FUNCTION_BLOCK SensorFQM
VAR_INPUT
END_VAR
VAR_OUTPUT
END_VAR
VAR_IN_OUT
	
END_VAR
VAR
	State:VisionState:= 0;
	SensorToPlc AT %I*:SensorToPlc;
	PlcToSensor AT %Q*:PlcToSensor;
	KeepAliveTimer:TON;
	
	RExec:R_TRIG;
	NextCycleResetFlags:BOOL;
	Results: ARRAY [0..7] OF REAL;
	
	//Single measurement
	RequestSingle:BOOL;
	TakePhoto:BOOL;
	TakePhotoFlag:R_TRIG;
	MeasureTimer:TON;
	MeasureTime:TIME;
	
	//Continuous measurement
	RequestStartCont:BOOL;
	RequestStopCont:BOOL;
	StopFromError:BOOL;
	ResponseTimer:TON;
	ResponseTime:TIME;
	FEnable:F_TRIG;
	
	LastResult:INT:=0;//0-Null, 1-Ok, 2-NG
	
	//Error Management
	RequestErrorCode:BOOL;
	LastError:DWORD;
END_VAR
VAR CONSTANT
	KeepAliveBit:INT:=24;
END_VAR

// Preparing Inputs
SensorToPlc.FLG:= SensorToPlc.VisionStatusFlag.0;
SensorToPlc.BUSY:= SensorToPlc.VisionStatusFlag.1;
SensorToPlc.READY:= SensorToPlc.VisionStatusFlag.2;
SensorToPlc.OR_Jud:= SensorToPlc.VisionStatusFlag.3;
SensorToPlc.RUN:= SensorToPlc.VisionStatusFlag.4;
SensorToPlc.ERR:= SensorToPlc.VisionStatusFlag.15;
SensorToPlc.GATE:= SensorToPlc.VisionStatusFlag.16;
//Change a bit every 500ms as Keep Alive bit
(*KeepAliveTimer(in:=NOT KeepAliveTimer.Q, pt:=T#1S);
IF KeepAliveTimer.Q THEN
	PlcToSensor.VisionControlFlag.24:= NOT PlcToSensor.VisionControlFlag.24;
END_IF*)

//Delete variables. Estado distinto de 999 para permitir modificar a mano en ese estado especial
IF State <> 999 THEN
	PlcToSensor.EXE:=FALSE;
	PlcToSensor.ERCLR:=FALSE;
	PlcToSensor.DSA:=FALSE;
	PlcToSensor.TRIG:=FALSE;
END_IF

//State machine
CASE State OF
	000: //Error. Por ahora se salta parada cuando hay error
		IF NOT SensorToPlc.ERR THEN
			State := 010;
		ELSE
			State := 001;
		END_IF
			
	001: //Checking errors
		//TODO: Revisar
		_prepareCommand(Command:= VisionCmd.GetLatestError);
		PlcToSensor.EXE := TRUE;
		IF SensorToPlc.FLG THEN
			PlcToSensor.EXE := FALSE;
			LastError:= SensorToPlc.VisionResponseData;
			State := 002;
		END_IF
	002: //Clear data
		_prepareCommand(VisionCmd.ClearDataOutputBuffer);
		PlcToSensor.EXE := TRUE;
		IF SensorToPlc.FLG THEN
			PlcToSensor.EXE := FALSE;
			State := 003;
		END_IF
	003: //Clear Error
		PlcToSensor.ERCLR:=TRUE;
		IF NOT SensorToPlc.ERR THEN
			PlcToSensor.ERCLR := FALSE;
			State := 010;
		END_IF
	010: //StandStill
		IF RequestSingle THEN
			LastError := 0; //Elimina ultimo error cuando se pasa a este estado
			State := 011;
		END_IF
		IF RequestStartCont AND NOT RequestSingle THEN
			State := 012;
		END_IF
		IF SensorToPlc.ERR THEN
			State := 001;
			
		END_IF
	011: //Switching to Single
		_prepareCommand(VisionCmd.StartSingle);
		PlcToSensor.EXE:=TRUE;
		IF SensorToPlc.FLG THEN
			PlcToSensor.EXE := FALSE;
			State := 030;
			LastResult:=0;
		END_IF
	012: //Switching to continuous
		_prepareCommand(VisionCmd.StartContinuous);
		PlcToSensor.EXE:=TRUE;
		IF SensorToPlc.FLG THEN
			PlcToSensor.EXE := FALSE;
			State := 020;
		END_IF
	020: //Continuous Measurement
		//Loop to request measurement
		IF SensorToPlc.GATE THEN
			ResponseTime:=ResponseTimer.ET;
			PlcToSensor.DSA := FALSE;
			ResponseTimer(in:=FALSE, pt:=T#10S);
		ELSIF NOT SensorToPLC.gate THEN
			ResponseTimer(in:=TRUE, pt:=T#10S);
			PlcToSensor.DSA := TRUE;
		END_IF
		//transitions
		IF SensorToPLC.ERR THEN
			PlcToSensor.EXE := FALSE;
			StopFromError:=TRUE;
			State := 021;
		END_IF 
		IF RequestStopCont THEN
			PlcToSensor.EXE := FALSE;
			State := 021;
		END_IF
	021: //Stopping continuous
	    _prepareCommand(VisionCmd.StopContinuous);
		PlcToSensor.EXE := TRUE;
		IF SensorToPLC.FLG THEN
			IF StopFromError THEN
				PlcToSensor.EXE :=FALSE;
				StopFromError:=FALSE;
				State := 001;
			ELSE
				State := 010;
			END_IF
			RequestStopCont := FALSE;
		END_IF
	030: // Single Measurement Ready
		
		IF TakePhoto THEN
			//Take photo and request
			PlcToSensor.TRIG:=TRUE;
			PlcToSensor.DSA:=TRUE;
			MeasureTimer(in:=FALSE);
			MeasureTimer(in:=TRUE, pt:=T#60s);
			State := 31;
		END_IF
		IF NOT RequestSingle THEN
			State := 010;
		END_IF
		IF SensorToPlc.ERR THEN
			State := 001;
			_prepareCommand(Command:= VisionCmd.GetLatestError);
			PlcToSensor.EXE := TRUE;
		END_IF
	031: // Single Measurement Taking photo
		PlcToSensor.DSA := TRUE; // Ojo, ya se activo en el ciclo anterior. no hay retardo de un ciclo.
		PlcToSensor.TRIG := TRUE;
		MeasureTimer(in:=TRUE);
		IF SensorToPLC.GATE THEN
			//TODO: Esto llega mas tarde que el dato. Revisar.
			IF SensorToPlc.OR_Jud THEN
				LastResult:=2;
			ELSE
				LastResult:=1;
			END_IF
			MeasureTime:=MeasureTimer.ET;
			MeasureTimer(in:=FALSE);
			State := 030;
			PlcToSensor.TRIG:=FALSE;
			PlcToSensor.DSA:=FALSE;
		END_IF
		IF SensorToPLC.ERR THEN
			State := 001;
		END_IF
END_CASE

//Update Flag Bits into DWORD
PlcToSensor.VisionControlFlag.0:= PlcToSensor.EXE;
PlcToSensor.VisionControlFlag.1:= PlcToSensor.TRIG;
PlcToSensor.VisionControlFlag.15:= PlcToSensor.ERCLR;
PlcToSensor.VisionControlFlag.16:= PlcToSensor.DSA;

METHOD PRIVATE _prepareCommand
VAR_INPUT
	Command:VisionCmd;
END_VAR
VAR
	
END_VAR
(* 
Command orders deliverable to camera.
See OMRON FQ-M Series Vision Sensor docs for information
*)
CASE Command OF
	VisionCmd.StartSingle: 				PlcToSensor.VisionCommand:= 16#00101010;
	VisionCmd.StartContinuous: 			PlcToSensor.VisionCommand:= 16#00101020;
	VisionCmd.StopContinuous: 			PlcToSensor.VisionCommand:= 16#00101030;
	VisionCmd.ClearValues: 				PlcToSensor.VisionCommand:= 16#00102010;
	VisionCmd.ClearDataOutputBuffer: 	PlcToSensor.VisionCommand:= 16#00102020;
	VisionCmd.Reset: 					PlcToSensor.VisionCommand:= 16#0010F010;
	VisionCmd.GetLatestError: 			PlcToSensor.VisionCommand:= 16#00205000;
END_CASE
END_METHOD

METHOD PUBLIC ContinuousShot : BOOL
VAR_INPUT
	Enable:BOOL; //Habilita el modo continuo. NOTA: Tendrá prioridad el modo único
END_VAR
VAR_OUTPUT
	Q:ARRAY [0..7] OF REAL;
END_VAR
FEnable(CLK:=Enable);
IF Enable THEN
	RequestStartCont:=TRUE;
	RequestStopCont:=FALSE;
END_IF
IF FEnable.Q THEN
	RequestStartCont:=FALSE;
	RequestStopCont:=TRUE;
	PlcToSensor.DSA:=FALSE;
	ResponseTimer(in:=FALSE);
END_IF

IF Enable THEN
//	IF SensorToPlc.GATE THEN
//		ResponseTime:=ResponseTimer.ET;
//		PlcToSensor.DSA := FALSE;
//		ResponseTimer(in:=FALSE, pt:=T#10S);
//	ELSIF NOT SensorToPLC.gate THEN
//		ResponseTimer(in:=TRUE, pt:=T#10S);
//		PlcToSensor.DSA := TRUE;
//	END_IF
;
END_IF

Q := SensorToPlc.VisionDataOutput;
END_METHOD

METHOD PUBLIC SingleShot : BOOL
VAR_INPUT
	Enable:BOOL;
	Execute:BOOL;
END_VAR
VAR_OUTPUT
	Active:BOOL;
	Measurement:BOOL;
	Ok:BOOL;
	Ng:BOOL;
	Q: ARRAY [0..7] OF REAL;
END_VAR
IF Enable THEN
	RequestSingle:=TRUE;
ELSE
	RequestSingle:=FALSE;
END_IF

TakePhotoFlag(clk:= Execute);
IF State = 030 THEN
	Active:=TRUE;
	IF TakePhotoFlag.Q THEN
		TakePhoto:=TRUE;
		Ok:=FALSE;
		Ng:=FALSE;
	END_IF
	CASE LastResult OF
		0: Ok:=FALSE; Ng:=FALSE; Measurement:=FALSE;
		1: Ok:=TRUE; Ng:=FALSE; Measurement:=TRUE;
		2: Ok:=FALSE; Ng:=TRUE; Measurement:= TRUE;
	END_CASE
	
ELSIF State = 031 THEN
	TakePhoto:=FALSE;
END_IF

Q := SensorToPlc.VisionDataOutput;
END_METHOD

END_FUNCTION_BLOCK

(* stored: Version 1.1.0.1, ProductVersion 3.1.4024.9
   POU SensorFQM: Id {8ea74fb3-e201-4806-8f67-b84ba6b734a0}, SpecialFunc None
   Method _prepareCommand: Id {a5013f73-e3c6-4216-beb5-427e6727c662}
   Method ContinuousShot: Id {7aa3080a-191c-450f-ad99-76e6e4f7b2ac}
   Method SingleShot: Id {87e13948-808e-4978-b44c-43911b4f1ae7} *)
